// TIA Portal project "Test_Fault_LowVoltage" (V14)

(* hardware
DEVICE "S7-1200 station_1"  S7-1200 Station
   slot 0: "Rack_0"  S7-1200 Rack  Rack  V1.0
   slot 1: "PLC_1"  CPU 1214C DC/DC/DC  6ES7 214-1AG40-0XB0  V4.2
DEVICE "HMI_1"  KTP700 Basic PN
   slot 0: "KTP700 Basic PN"  KTP700 Basic PN  6AV2 123-2GB03-0AX0  14.0.1.0
   slot 1: "HMI_RT_1"  KTP700 Basic PN  6AV2 123-2GB03-0AX0  14.0.1.0
   slot 5: "HMI_1.IE_CP_1"  PROFINET Interface  14.0.1.0
      slot 1: "PROFINET Interface_1"  PROFINET Interface
         slot 1: "Port_1"  Port
*)

// ===== PLC "PLC_1"  CPU 1214C DC/DC/DC =====

VAR_GLOBAL   // PLC tag table "Default tag table"
   "Normal" AT %Q0.0 : Bool;
   "Low_Volt" AT %Q0.1 : Bool;
   "Short_Circuit" AT %Q0.2 : Bool;
   "Freq_Fault" AT %Q0.3 : Bool;
   "Open_Circuit" AT %Q0.4 : Bool;
   "Overload" AT %Q0.5 : Bool;
   "illegal_load" AT %Q0.6 : Bool;
   "Poor_PF" AT %Q0.7 : Bool;
   "Clock_Byte" AT %MB0 : Byte;
   "Clock_10Hz" AT %M0.0 : Bool;
   "Clock_5Hz" AT %M0.1 : Bool;
   "Clock_2.5Hz" AT %M0.2 : Bool;
   "Clock_2Hz" AT %M0.3 : Bool;
   "Clock_1.25Hz" AT %M0.4 : Bool;
   "Clock_1Hz" AT %M0.5 : Bool;
   "Clock_0.625Hz" AT %M0.6 : Bool;
   "Clock_0.5Hz" AT %M0.7 : Bool;
END_VAR

VAR_GLOBAL   // PLC tag table "HOLD_REG"
   "40001" AT %MW100 : Word;
   "40002" AT %MW102 : Word;
   "40003" AT %MW104 : Word;
   "40004" AT %MW106 : Word;
   "40005" AT %MW108 : Word;
   "40006" AT %MW110 : Word;
   "40007" AT %MW112 : Word;
   "40008" AT %MW114 : Word;
   "40009" AT %MW116 : Word;
   "40010" AT %MW118 : Word;
   "40011" AT %MW120 : Word;
   "40012" AT %MW122 : Word;
   "40013" AT %MW124 : Word;
   "40014" AT %MW126 : Word;
   "40015" AT %MW128 : Word;
   "40016" AT %MW130 : Word;
   "40017" AT %MW132 : Word;
   "40018" AT %MW134 : Word;
   "40019" AT %MW136 : Word;
   "40020" AT %MW138 : Word;
END_VAR

DATA_BLOCK "Input_DB"   // DB1
{ S7_Optimized_Access := 'TRUE' }
VERSION : 0.1
   VAR
      "Send_Frequency [Hz]" : DInt := 50;
      "Send_Voltage [V]" : DInt := 230;
      "Send_Current [mA]" : DInt := 23;
      "Send_Energy [KWh]" : DInt;
      "Send_ActivePwr [W]" : DInt := 900;
      "Send_ReactivePwr [KVAr]" : DInt;
      Send_PwrFactor : DInt := 800;
      "Recv_Frequency [Hz]" : DInt := 50;
      "Recv_Voltage [V]" : DInt := 230;
      "Recv_Current [mA]" : DInt := 23;
      "Recv_Energy [KWh]" : DInt;
      "Recv_ActivePwr [W]" : DInt := 900;
      "Recv_ReactivePwr [KVAr]" : DInt;
      Recv_PwrFactor : DInt := 800;
   END_VAR
BEGIN
END_DATA_BLOCK

DATA_BLOCK "Fault_DB"   // DB2
{ S7_Optimized_Access := 'TRUE' }
VERSION : 0.1
   VAR
      None : Bool;
      Low_Voltage : Bool;
      Short_Circuit : Bool;
      Freq_fault : Bool;
      Open_Circuit : Bool;
      High_Voltage : Bool;
      Overload : Bool;
      Illegal_Load : Bool;
      Poor_PF : Bool;
   END_VAR
BEGIN
END_DATA_BLOCK

DATA_BLOCK "Cond_DB"   // DB3
{ S7_Optimized_Access := 'TRUE' }
VERSION : 0.1
   VAR
      Recv_PwrLimit : Int := 1000;
      error_ActivePwr : Int;
      Psend_10percent : Int;
      PwrFactor_Limit : Int := 800;
      Freq_LowerLImit : Int := 4750;
      Freq_UpperLimit : Int := 5250;
      Current_Limit : Int := 10;
      Vsend_5percent : Int := 220;
      Vsend_10percent : Int := 208;
      Vsend_High : Int := 242;
   END_VAR
BEGIN
END_DATA_BLOCK

DATA_BLOCK "Modbus_Client_DB"   // DB9
{ S7_Optimized_Access := 'TRUE' }
VERSION : 0.1
   VAR
      Done : Bool;
      Busy : Bool;
      Error : Bool;
      Status : Word;
      ConnectParam : TCON_IP_v4;
   END_VAR
BEGIN
   ConnectParam.InterfaceId := 64;
   ConnectParam.ID := 16#2;
   ConnectParam.ActiveEstablished := true;
   ConnectParam.RemoteAddress.ADDR[1] := 192;
   ConnectParam.RemoteAddress.ADDR[2] := 168;
   ConnectParam.RemoteAddress.ADDR[3] := 0;
   ConnectParam.RemoteAddress.ADDR[4] := 107;
   ConnectParam.RemotePort := 502;
   ConnectParam.LocalPort := 0;
END_DATA_BLOCK

ORGANIZATION_BLOCK "Main"   // OB1, LAD, ProgramCycle
TITLE = "Main Program Sweep (Cycle)"
{ S7_Optimized_Access := 'TRUE' }
VERSION : 0.1
   VAR_INPUT
      Initial_Call : Bool;   // Initial call of this OB
      Remanence : Bool;   // =True, if remanent data are available
   END_VAR
   VAR_TEMP
      Freq_Fault : Bool;
   END_VAR
BEGIN

REGION Network 1: Detect Fault
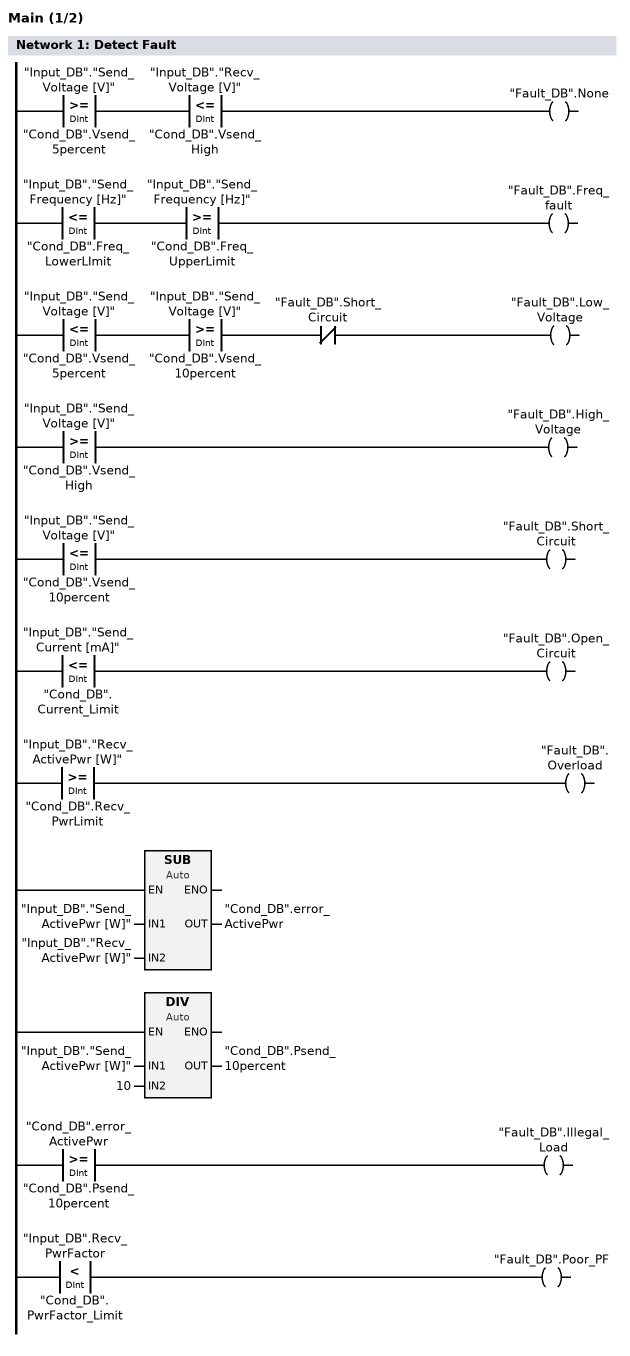
   RUNG wire#powerrail
      { S7_Templates := "SrcType := DInt" } GE_Contact(in1 := "Input_DB"."Send_Voltage [V]", in2 := "Cond_DB".Vsend_5percent)
      { S7_Templates := "SrcType := DInt" } LE_Contact(in1 := "Input_DB"."Recv_Voltage [V]", in2 := "Cond_DB".Vsend_High)
      Coil( "Fault_DB".None )
   END_RUNG
   RUNG wire#powerrail
      { S7_Templates := "SrcType := DInt" } LE_Contact(in1 := "Input_DB"."Send_Frequency [Hz]", in2 := "Cond_DB".Freq_LowerLImit)
      { S7_Templates := "SrcType := DInt" } GE_Contact(in1 := "Input_DB"."Send_Frequency [Hz]", in2 := "Cond_DB".Freq_UpperLimit)
      Coil( "Fault_DB".Freq_fault )
   END_RUNG
   RUNG wire#powerrail
      { S7_Templates := "SrcType := DInt" } LE_Contact(in1 := "Input_DB"."Send_Voltage [V]", in2 := "Cond_DB".Vsend_5percent)
      { S7_Templates := "SrcType := DInt" } GE_Contact(in1 := "Input_DB"."Send_Voltage [V]", in2 := "Cond_DB".Vsend_10percent)
      I_Contact( "Fault_DB".Short_Circuit )
      Coil( "Fault_DB".Low_Voltage )
   END_RUNG
   RUNG wire#powerrail
      { S7_Templates := "SrcType := DInt" } GE_Contact(in1 := "Input_DB"."Send_Voltage [V]", in2 := "Cond_DB".Vsend_High)
      Coil( "Fault_DB".High_Voltage )
   END_RUNG
   RUNG wire#powerrail
      { S7_Templates := "SrcType := DInt" } LE_Contact(in1 := "Input_DB"."Send_Voltage [V]", in2 := "Cond_DB".Vsend_10percent)
      Coil( "Fault_DB".Short_Circuit )
   END_RUNG
   RUNG wire#powerrail
      { S7_Templates := "SrcType := DInt" } LE_Contact(in1 := "Input_DB"."Send_Current [mA]", in2 := "Cond_DB".Current_Limit)
      Coil( "Fault_DB".Open_Circuit )
   END_RUNG
   RUNG wire#powerrail
      { S7_Templates := "SrcType := DInt" } GE_Contact(in1 := "Input_DB"."Recv_ActivePwr [W]", in2 := "Cond_DB".Recv_PwrLimit)
      Coil( "Fault_DB".Overload )
   END_RUNG
   RUNG wire#powerrail
      Sub(in1 := "Input_DB"."Send_ActivePwr [W]", in2 := "Input_DB"."Recv_ActivePwr [W]", out => "Cond_DB".error_ActivePwr)
   END_RUNG
   RUNG wire#powerrail
      Div(in1 := "Input_DB"."Send_ActivePwr [W]", in2 := 10, out => "Cond_DB".Psend_10percent)
   END_RUNG
   RUNG wire#powerrail
      { S7_Templates := "SrcType := DInt" } GE_Contact(in1 := "Cond_DB".error_ActivePwr, in2 := "Cond_DB".Psend_10percent)
      Coil( "Fault_DB".Illegal_Load )
   END_RUNG
   RUNG wire#powerrail
      { S7_Templates := "SrcType := DInt" } LT_Contact(in1 := "Input_DB".Recv_PwrFactor, in2 := "Cond_DB".PwrFactor_Limit)
      Coil( "Fault_DB".Poor_PF )
   END_RUNG
   // the same network as SCL:
   "Fault_DB".None := ("Input_DB"."Send_Voltage [V]" >= "Cond_DB".Vsend_5percent) AND ("Input_DB"."Recv_Voltage [V]" <= "Cond_DB".Vsend_High);
   "Fault_DB".Freq_fault := ("Input_DB"."Send_Frequency [Hz]" <= "Cond_DB".Freq_LowerLImit) AND ("Input_DB"."Send_Frequency [Hz]" >= "Cond_DB".Freq_UpperLimit);
   "Fault_DB".Low_Voltage := ("Input_DB"."Send_Voltage [V]" <= "Cond_DB".Vsend_5percent) AND ("Input_DB"."Send_Voltage [V]" >= "Cond_DB".Vsend_10percent) AND NOT "Fault_DB".Short_Circuit;
   "Fault_DB".High_Voltage := "Input_DB"."Send_Voltage [V]" >= "Cond_DB".Vsend_High;
   "Fault_DB".Short_Circuit := "Input_DB"."Send_Voltage [V]" <= "Cond_DB".Vsend_10percent;
   "Fault_DB".Open_Circuit := "Input_DB"."Send_Current [mA]" <= "Cond_DB".Current_Limit;
   "Fault_DB".Overload := "Input_DB"."Recv_ActivePwr [W]" >= "Cond_DB".Recv_PwrLimit;
   "Cond_DB".error_ActivePwr := "Input_DB"."Send_ActivePwr [W]" - "Input_DB"."Recv_ActivePwr [W]";
   "Cond_DB".Psend_10percent := "Input_DB"."Send_ActivePwr [W]" / 10;
   "Fault_DB".Illegal_Load := "Cond_DB".error_ActivePwr >= "Cond_DB".Psend_10percent;
   "Fault_DB".Poor_PF := "Input_DB".Recv_PwrFactor < "Cond_DB".PwrFactor_Limit;
END_REGION

REGION Network 2: Display Fault
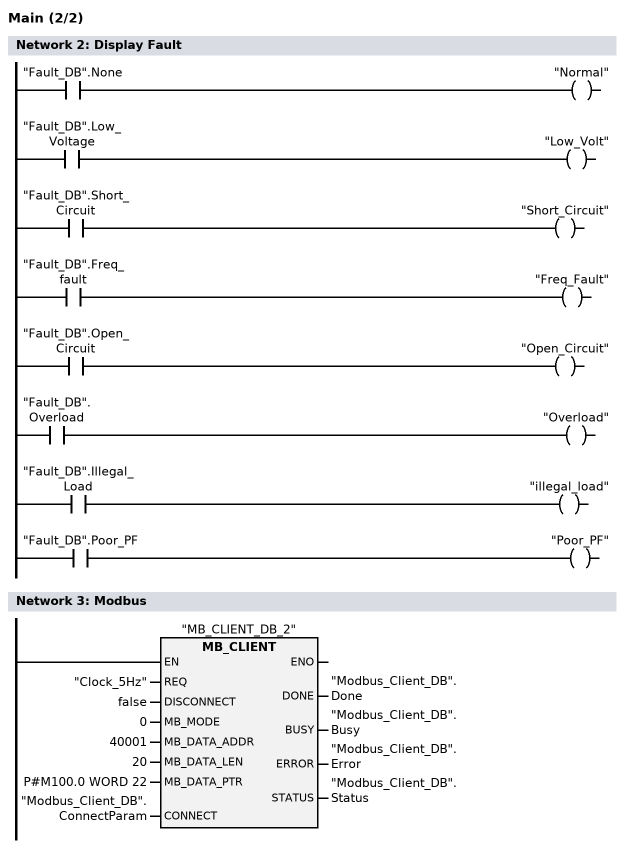
   RUNG wire#powerrail
      Contact( "Fault_DB".None )
      Coil( "Normal" )
   END_RUNG
   RUNG wire#powerrail
      Contact( "Fault_DB".Low_Voltage )
      Coil( "Low_Volt" )
   END_RUNG
   RUNG wire#powerrail
      Contact( "Fault_DB".Short_Circuit )
      Coil( "Short_Circuit" )
   END_RUNG
   RUNG wire#powerrail
      Contact( "Fault_DB".Freq_fault )
      Coil( "Freq_Fault" )
   END_RUNG
   RUNG wire#powerrail
      Contact( "Fault_DB".Open_Circuit )
      Coil( "Open_Circuit" )
   END_RUNG
   RUNG wire#powerrail
      Contact( "Fault_DB".Overload )
      Coil( "Overload" )
   END_RUNG
   RUNG wire#powerrail
      Contact( "Fault_DB".Illegal_Load )
      Coil( "illegal_load" )
   END_RUNG
   RUNG wire#powerrail
      Contact( "Fault_DB".Poor_PF )
      Coil( "Poor_PF" )
   END_RUNG
   // the same network as SCL:
   "Normal" := "Fault_DB".None;
   "Low_Volt" := "Fault_DB".Low_Voltage;
   "Short_Circuit" := "Fault_DB".Short_Circuit;
   "Freq_Fault" := "Fault_DB".Freq_fault;
   "Open_Circuit" := "Fault_DB".Open_Circuit;
   "Overload" := "Fault_DB".Overload;
   "illegal_load" := "Fault_DB".Illegal_Load;
   "Poor_PF" := "Fault_DB".Poor_PF;
END_REGION

REGION Network 3: Modbus
   "MB_CLIENT_DB_2"(REQ := "Clock_5Hz",   // MB_CLIENT
                    DISCONNECT := false,
                    MB_MODE := 0,
                    MB_DATA_ADDR := 40001,
                    MB_DATA_LEN := 20,
                    MB_DATA_PTR := P#M100.0 WORD 22,
                    CONNECT := "Modbus_Client_DB".ConnectParam,
                    DONE => "Modbus_Client_DB".Done,
                    BUSY => "Modbus_Client_DB".Busy,
                    ERROR => "Modbus_Client_DB".Error,
                    STATUS => "Modbus_Client_DB".Status);
END_REGION
END_ORGANIZATION_BLOCK

(* ===== HMI "HMI_RT_1" =====
system functions are stored by id; their names below are inferred from use
connection "HMI_Connection_1": ETHERNET, SMART_S7_1200_OMS

HMI tags "Default tag table"
   "Tag_ScreenNumber" : UInt, internal
   "Input_DB_Send_Frequency [Hz]" : DInt = PLC Input_DB."Send_Frequency [Hz]", 1 s
   "Input_DB_Send_Voltage [V]" : DInt = PLC Input_DB."Send_Voltage [V]", 1 s
   "Input_DB_Send_Energy [KWh]" : DInt = PLC Input_DB."Send_Energy [KWh]", 1 s
   "Normal" : Bool = PLC Normal AT %Q0.0, 1 s
   "Low_Volt" : Bool = PLC Low_Volt AT %Q0.1, 1 s
   "Overload" : Bool = PLC Freq_Fault AT %Q0.3, 1 s
   "Short_Circuit" : Bool = PLC Short_Circuit AT %Q0.2, 1 s
   "Input_DB_Send_ActivePwr [W]" : DInt = PLC Input_DB."Send_ActivePwr [W]", 1 s
   "Input_DB_Send_Current [A]" : DInt = PLC Input_DB."Send_Current [mA]", 1 s
   "Input_DB_Send_PwrFactor" : DInt = PLC Input_DB.Send_PwrFactor, 1 s
   "Input_DB_Recv_Frequency [Hz]" : DInt = PLC Input_DB."Recv_Frequency [Hz]", 1 s
   "Input_DB_Recv_Voltage [V]" : DInt = PLC Input_DB."Recv_Voltage [V]", 1 s
   "Input_DB_Recv_Current [A]" : DInt = PLC Input_DB."Recv_Current [mA]", 1 s
   "Input_DB_Recv_ActivePwr [W]" : DInt = PLC Input_DB."Recv_ActivePwr [W]", 1 s
   "Input_DB_Recv_PwrFactor" : DInt = PLC Input_DB.Recv_PwrFactor, 1 s
   "Fault_DB_Low_Voltage" : Bool = PLC Fault_DB.Low_Voltage, 1 s
   "Fault_DB_Short_Circuit" : Bool = PLC Fault_DB.Short_Circuit, 1 s
   "Fault_DB_Open_Circuit" : Bool = PLC Fault_DB.Open_Circuit, 1 s
   "Fault_DB_Poor_PF" : Bool = PLC Fault_DB.Poor_PF, 1 s
   "Fault_DB_Overload" : Bool = PLC Fault_DB.Overload, 1 s
   "Fault_DB_Illegal_Load" : Bool = PLC Fault_DB.Illegal_Load, 1 s

Template "Template_1" 800x480
   Button "Exit" at 714,429 size 71x50; TextOff 'Exit'; PictureOff "ExitRuntime_KTP700_Basic_PN_TR"; PictureOn "ExitRuntime_KTP700_Basic_PN_TR"
      on Release: StopRuntime(0)
   Button "Template_Button" at 614,429 size 71x50; TextOff 'Text'
   Button "Template_Button_1" at 514,429 size 71x50; TextOff 'Text'
   Button "Template_Button_2" at 414,429 size 71x50; TextOff 'Text'
   Button "Template_Button_3" at 314,429 size 71x50; TextOff 'Text'
   Button "Template_Button_4" at 214,429 size 71x50; TextOff 'Text'
   Button "Alarms" at 114,429 size 71x50; TextOff 'Alarms'; PictureOff "AlarmDisplay_KTP700_Basic_PN_TR"; PictureOn "AlarmDisplay_KTP700_Basic_PN_TR"
      on Release: function_ef3f5d25("Alarm window_Unacknowledged", -1)
   Button "Start screen" at 14,429 size 71x50; TextOff 'Start screen'; PictureOff "NavigateHome_KTP700_Basic_PN_TR"; PictureOn "NavigateHome_KTP700_Basic_PN_TR"
      on Release: ActivateScreen("Root screen", 0)
   DateTimeField "HmiScreenItemData" at 695,25 size 105x25
   DateTimeField "HmiScreenItemData_1" at 695,0 size 105x25
   GraphicView "Logo" at 0,0 size 91x51; Picture "Logo of HMI_1"

screen "Root screen" 800x480, template "Template_1"
   on GenerateScreen: SetTag("Tag_ScreenNumber", 1)
   TextField "HmiScreenItemData" at 80,225 size 640x25; Text 'Welcome to HMI_1 (KTP700 Basic+ PN)!'

screen "Screen_1" 800x480
   GraphicView "Graphic view_1" at 0,0 size 799x480; Picture "600px-UK_Fin_Flash_low_visiability.svg"
   TextField "Text field_1" at 39,59 size 115x32; Text 'SENDING'
   TextField "Text field_2" at 262,59 size 138x32; Text 'RECEIVING'
   TextField "Text field_3" at 191,111 size 40x37; Text 'Hz'
   TextField "Text field_4" at 185,173 size 73x37; Text 'Volts'
   TextField "Text field_5" at 168,234 size 106x37; Text 'mAmps'
   TextField "Text field_6" at 185,297 size 33x37; Text 'W'
   TextField "Text field_7" at 185,364 size 39x37; Text 'PF'
   IOField "I/O field_1" at 45,111 size 96x32; FormatPattern 999
      ProcessValue <- "Input_DB_Send_Frequency [Hz]"
   IOField "I/O field_2" at 46,173 size 96x32; FormatPattern 99999
      ProcessValue <- "Input_DB_Send_Voltage [V]"
   IOField "I/O field_3" at 45,298 size 96x32; FormatPattern 99999
      ProcessValue <- "Input_DB_Send_ActivePwr [W]"
   DateTimeField "Date/time field_1" at 115,422 size 211x24
   TextField "Text field_8" at 175,12 size 484x34; Text 'Power Distribution Monitoring System'
   Circle "Circle_1" at 419,75 size 66x66
      Appearance <- "Normal"
   Circle "Circle_2" at 419,195 size 66x66
      Appearance <- "Fault_DB_Open_Circuit"
   Circle "Circle_3" at 558,71 size 66x66
      Appearance <- "Fault_DB_Low_Voltage"
   TextField "Text field_9" at 417,150 size 76x23; Text 'NORMAL'
   TextField "Text field_10" at 524,149 size 129x23; Text 'LOW VOLTAGE'
   TextField "Text field_11" at 400,263 size 131x23; Text 'OPEN CIRCUIT'
   Circle "Circle_4" at 558,197 size 66x66
      Appearance <- "Fault_DB_Short_Circuit"
   TextField "Text field_12" at 532,262 size 143x23; Text 'SHORT CIRCUIT'
   IOField "I/O field_4" at 45,235 size 96x32; FormatPattern 999
      ProcessValue <- "Input_DB_Send_Current [A]"
   IOField "I/O field_5" at 45,365 size 96x32; FormatPattern 999
      ProcessValue <- "Input_DB_Send_PwrFactor"
   IOField "I/O field_6" at 291,106 size 96x37; FormatPattern 999
      ProcessValue <- "Input_DB_Recv_Frequency [Hz]"
   IOField "I/O field_7" at 290,167 size 98x39; FormatPattern 99999
      ProcessValue <- "Input_DB_Recv_Voltage [V]"
   IOField "I/O field_8" at 289,233 size 98x39; FormatPattern 999
      ProcessValue <- "Input_DB_Recv_Current [A]"
   IOField "I/O field_9" at 290,300 size 97x38; FormatPattern 99999
      ProcessValue <- "Input_DB_Recv_ActivePwr [W]"
   IOField "I/O field_10" at 289,357 size 101x45; FormatPattern 999
      ProcessValue <- "Input_DB_Recv_PwrFactor"
   Circle "Circle_5" at 419,297 size 66x66
      Appearance <- "Fault_DB_Illegal_Load"
   TextField "Text field_13" at 403,364 size 123x23; Text 'ILLEGAL LOAD'
   Circle "Circle_6" at 701,195 size 66x66
      Appearance <- "Fault_DB_Overload"
   TextField "Text field_14" at 688,261 size 95x23; Text 'OVERLOAD'
   Circle "Circle_7" at 558,297 size 66x66
      Appearance <- "Fault_DB_Poor_PF"
   TextField "Text field_15" at 558,365 size 77x23; Text 'POOR PF'
   Circle "Circle_8" at 701,71 size 66x66
      Appearance <- "Short_Circuit"
   TextField "Text field_16" at 677,149 size 109x23; Text 'FREQUENCY'
*)